Fanuc KAREL source: scn_new.kl

PROGRAM scn_new
%NOBUSYLAMP
%NOLOCKGROUP

%include defaultcell.klt
define_scan_object(SCANNING_OBJECT_NAME,SCANNING_CNFG)

BEGIN
	new
END scn_new
